FUNCTION_BLOCK M2TiltYAxis EXTENDS SM_M2TiltYAxis
VAR_INPUT
END_VAR
VAR_OUTPUT
END_VAR
VAR
    _lastRawValue : INT;
END_VAR


IF powered THEN
    _lastRawValue := SUPER^.position.rawValue;
ELSE
   SUPER^.position.rawValue := _lastRawValue;
END_IF

statuses.healthStatus(isGood := TRUE);

SUPER^(config := SUPER^.config, axisConfig := SUPER^.axisConfig);

END_FUNCTION_BLOCK

(* stored: Version 1.1.0.1, ProductVersion 3.1.4018.5
   POU M2TiltYAxis: Id {ec3d2749-ca8c-4f04-9ebb-21fdf51b178f}, SpecialFunc None *)
